FUNCTION rotY : mat3d
VAR_IN_OUT CONSTANT
	i_mat : Mat3d;
	i_ang : LREAL;
END_VAR
VAR
	rot :Mat3d := g_eye3d;
END_VAR

rot[1,1]:=COS(i_ang);
rot[3,3]:=rot[1,1];
rot[1,3]:=SIN(i_ang);
rot[3,1]:=-rot[1,3];
rotY := mat3Mat3(i_mat, rot);

END_FUNCTION

(* stored: Version 1.1.0.1, ProductVersion 3.1.4024.12
   POU rotY: Id {4642df8a-62fa-4796-b707-eab077d12800}, SpecialFunc None *)
